INTERFACE I_RpcSynchronousReplyReadyToSend

METHOD PUBLIC Send
END_METHOD

END_INTERFACE

(* stored: Version 1.1.0.1, ProductVersion 3.1.4024.12
   Itf I_RpcSynchronousReplyReadyToSend: Id {2c9d43c2-32f4-4514-b001-a2923f45c572}
   Method Send: Id {c44ba08e-7280-4b08-b8f3-63445a092ff4} *)
